PROGRAM MAIN
VAR
	el2008: FB_EL8DO;
	outRefs: st_OutputNums;
	outs: ARRAY [1..8] OF BOOL;
END_VAR

el2008(outputRef:= outRefs, outputs:=outs );

END_PROGRAM

(* stored: Version 1.1.0.1
   POU MAIN: Id {9b50dab5-b168-4e01-8e83-028d1b870d14}, SpecialFunc None *)
